(* PLC project Unnamed, Unknown Unnamed 1 *)
(* stored: creationDateTime 2025-11-19T16:42:43, modificationDateTime 2025-11-19T18:10:22 *)

PROGRAM task1
  VAR
    DOWN_Stop AT %IX0.1 : BOOL;  (* Will Turn OFF the LED *)
  END_VAR
  VAR
    Latch : BOOL;  (* Latch Bit Instruction *)
  END_VAR
  VAR
    UP_Start AT %IX0.0 : BOOL;  (* Will Turn ON the LED *)
    LED AT %QX0.0 : BOOL;  (* Output indicator for Latch_Unlatch Program *)
  END_VAR

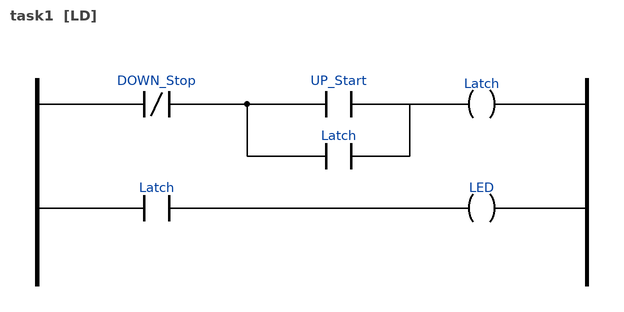
(* LD diagram, written out as Structured Text *)
Latch := NOT DOWN_Stop AND (UP_Start OR Latch);
LED := Latch;
END_PROGRAM

CONFIGURATION Config0
  RESOURCE Res0 ON PLC
    TASK task0(INTERVAL := T#20ms, PRIORITY := 0);
    PROGRAM instance0 WITH task0 : task1;
  END_RESOURCE
END_CONFIGURATION
